INTERFACE INTERNAL I_EntityNode EXTENDS I_Debug

PROPERTY INTERNAL _FirstComp : I_Component
GET
END_GET
SET
END_SET
END_PROPERTY

PROPERTY INTERNAL _LastComp : I_Component
GET
END_GET
SET
END_SET
END_PROPERTY

PROPERTY INTERNAL _Next : I_Entity
GET
END_GET
SET
END_SET
END_PROPERTY

PROPERTY INTERNAL _Prev : I_Entity
GET
END_GET
SET
END_SET
END_PROPERTY

PROPERTY INTERNAL _Size : UDINT
GET
END_GET
SET
END_SET
END_PROPERTY

PROPERTY INTERNAL _State : _EntityState
GET
END_GET
SET
END_SET
END_PROPERTY

(*
Description: Retrieves a previous component before the inputted one or last component if referenced value is 0.
Returns:
- Ok - Returns upon success, updates referenced value with new component.
- Err.InvRef - Invalid output reference.
- Err.ItfEq - Provided interface pointer doesn't belong to the queried entity. Nulls reference.
- Err.NotFound - The entity doesn't contain any components. Nulls reference.
- Err.End - No more components. Nulls reference.
*)
METHOD GetNextComp : Result
VAR_INPUT
	iOut		: REFERENCE TO I_Component;
END_VAR
END_METHOD

(*
Description: Retrieves a previous component before the inputted one or last component if referenced value is 0.
Returns:
- Ok - Returns upon success, updates referenced value with new component.
- Err.InvRef - Invalid output reference.
- Err.ItfEq - Provided interface pointer doesn't belong to the queried entity. Nulls reference.
- Err.NotFound - The entity doesn't contain any components. Nulls reference.
- Err.End - No more components. Nulls reference.
*)
METHOD GetPrevComp : Result
VAR_INPUT
	iOut		: REFERENCE TO I_Component;
END_VAR
END_METHOD

(*
Provides the size of the entity, indicating the number of components it manages.  
Note: For internal logic purposes, this value is incremented by one beyond the actual component count.
*)
PROPERTY Size : UDINT
GET
END_GET
END_PROPERTY

END_INTERFACE

(* stored: Version 1.1.0.1
   Itf I_EntityNode: Id {c69b9ec4-3971-4258-8ff6-b55228e1d9e3}
   Folder _: Id {da71af14-1425-4366-a03a-2e7575b43e6a}
   Property _FirstComp: Id {02fbe986-1bdd-415d-bb4c-ff100c6f2cf1}
   Get Get: Id {2975002c-0cdc-4aa1-b5e9-acee65f8547b}
   Set Set: Id {e87ade3c-21f3-4b70-b95e-77e6bcd74721}
   Property _LastComp: Id {c1e4c03f-9fb7-4237-84de-642f771cf470}
   Get Get: Id {8b32a67b-247b-4f83-a33d-10a5ecb0f5fc}
   Set Set: Id {5c8f06ab-af96-49c6-9975-37dcc2f94c35}
   Property _Next: Id {e667f3fa-d3de-4c97-8db5-27fcacd5a238}
   Get Get: Id {4c57db17-30bf-4e86-8e10-77f9968b4503}
   Set Set: Id {fcca1456-e6a2-453d-88ef-a0f9404dce8c}
   Property _Prev: Id {f2f7accb-05a3-40d7-b5a4-49e3057c46d0}
   Get Get: Id {926a06b1-a5bf-4b7a-bece-89e9ea4eaffa}
   Set Set: Id {073adfac-a98c-4de6-a2f2-f331fad5a6e2}
   Property _Size: Id {442dacda-2b3b-44ad-97d6-2d86502474fc}
   Get Get: Id {bbf338cc-44ea-4dd3-872c-937a773a321d}
   Set Set: Id {e1783e5c-5753-41d7-a64e-80405fd8388d}
   Property _State: Id {4bbace86-cd64-4c27-8035-1596b4824ba1}
   Get Get: Id {91d63009-bbdd-4b02-b445-6bd121e4fccc}
   Set Set: Id {77096148-17ba-4b28-bc31-3a9dfedc8dd8}
   Method GetNextComp: Id {afbd579f-fd8e-4b2e-abcf-16fd7b88f3d9}
   Method GetPrevComp: Id {74204c05-ffc4-4fb9-8e9e-cba9dc367ab1}
   Property Size: Id {566027c5-cdc2-4034-8eb4-a311c8741cd8}
   Get Get: Id {717b31d4-ecc7-4a6c-bc4d-7f7fd087a1fc} *)
